GLOBALCONSTANTS Computers (* Global constants *)
  (* Standard: 61499-1 *)
  (* Version 1.0, 2023-10-22, franz *)
  VAR_GLOBAL CONSTANT
    C_LO : WSTRING := "localhost:61499";
    C_ET : WSTRING := "192.168.5.1:61499";
    C_ST : WSTRING := "192.168.4.1:61499";
    C_00 : WSTRING := "192.168.4.1:61499";
  END_VAR
END_GLOBALCONSTANTS
